(*!
<summary>{attribute 'OPC.UA.DA.Access' := '1'}</summary>
*)

{attribute 'no_explicit_call' := 'do not call this function block directly'}
FUNCTION_BLOCK ABSTRACT ProgramTransition EXTENDS ToolkitObject IMPLEMENTS IAction
VAR_OUTPUT
	
	//Timeout : TIME := T#3S;
END_VAR
VAR
	{attribute 'OPC.UA.DA' := '0'}
	_Busy : BOOL;
	{attribute 'OPC.UA.DA' := '0'}
	_Done : BOOL;
	{attribute 'OPC.UA.DA' := '0'}
	_Error : BOOL;
	{attribute 'OPC.UA.DA' := '0'}
	_StateMachine : REFERENCE TO FiniteStateMachine;
END_VAR

{attribute 'monitoring' := 'call'}
{attribute 'OPC.UA.DA.Property' := '1'}
{attribute 'OPC.UA.DA.Access' := '1'}
PROPERTY Busy : BOOL
GET
Busy := _Busy;
END_GET
END_PROPERTY

METHOD Cancel
IF _Busy THEN
	_Busy := FALSE;	
END_IF
END_METHOD

{attribute 'monitoring' := 'call'}
{attribute 'OPC.UA.DA.Property' := '1'}
{attribute 'OPC.UA.DA.Access' := '1'}
PROPERTY ABSTRACT Cause : STRING
GET
END_GET
END_PROPERTY

{attribute 'monitoring' := 'call'}
{attribute 'OPC.UA.DA.Property' := '1'}
{attribute 'OPC.UA.DA.Access' := '1'}
PROPERTY Done : BOOL
GET
Done := _Done;
END_GET
END_PROPERTY

{attribute 'monitoring' := 'call'}
{attribute 'OPC.UA.DA.Property' := '1'}
{attribute 'OPC.UA.DA.Access' := '1'}
PROPERTY Error : BOOL
GET
Error := _Error;
END_GET
END_PROPERTY

METHOD Execute
_Busy := FALSE;
_Done := TRUE;
_Error := FALSE;
END_METHOD

{attribute 'monitoring' := 'call'}
{attribute 'OPC.UA.DA.Property' := '1'}
{attribute 'OPC.UA.DA.Access' := '1'}
PROPERTY ABSTRACT FromState : STRING
GET
END_GET
END_PROPERTY

METHOD Initialize
VAR_INPUT
	stateMachine : REFERENCE TO FiniteStateMachine;
END_VAR
IF NOT __ISVALIDREF(_StateMachine) THEN
	//exceptionFactory.ThrowException(__POSITION(), "programStateMachine is NULL");
END_IF

_StateMachine REF= stateMachine;
END_METHOD

{attribute 'monitoring' := 'call'}
{attribute 'OPC.UA.DA.Property' := '1'}
{attribute 'OPC.UA.DA.Access' := '1'}
PROPERTY Initialized : BOOL
GET
Initialized := __ISVALIDREF(_StateMachine);
END_GET
END_PROPERTY

{attribute 'monitoring' := 'call'}
PROPERTY LastException : REFERENCE TO Exception
GET
LastException REF= _LastException;
END_GET
END_PROPERTY

{attribute 'monitoring' := 'call'}
{attribute 'OPC.UA.DA.Property' := '1'}
{attribute 'OPC.UA.DA.Access' := '1'}
PROPERTY ABSTRACT Name : STRING
GET
END_GET
END_PROPERTY

METHOD Start
_Busy := FALSE;
_Done := TRUE;
_Error := FALSE;
END_METHOD

{attribute 'monitoring' := 'call'}
{attribute 'OPC.UA.DA.Property' := '1'}
{attribute 'OPC.UA.DA.Access' := '1'}
PROPERTY ABSTRACT ToState : STRING
GET
END_GET
END_PROPERTY

END_FUNCTION_BLOCK

(* stored: Version 1.1.0.1
   POU ProgramTransition: Id {6b59fb44-7d1e-410e-98ab-ba5c7025a4ba}, SpecialFunc None
   Property Busy: Id {b83feb43-f5ff-4bb3-87f5-84ead7a6b586}
   Get Get: Id {ea3ffc98-f880-4a1b-896f-a5358b6fb59b}
   Method Cancel: Id {f4d9f4ec-d47f-4802-b147-e47fb819abd8}
   Property Cause: Id {c9f3fd3d-674d-4611-85bc-8ec662b2c076}
   Get Get: Id {d1aac4fd-1f0a-4a8b-b9e2-9063ada794c0}
   Property Done: Id {c524e9f7-2d5a-4c7e-adac-dc51846488f5}
   Get Get: Id {be929d92-172b-4242-b667-f55e8250fbc4}
   Property Error: Id {fe37c4cb-37ea-43e6-a810-94afe137c611}
   Get Get: Id {4651eb3c-608a-4238-8ae6-8da6f587b31e}
   Method Execute: Id {1585fa56-5dfa-4194-aa2d-51a9ac8d90c2}
   Property FromState: Id {140a3845-da88-47be-b906-08a2791f1ee0}
   Get Get: Id {28420d79-259f-472e-a390-fe4adef5a6f9}
   Method Initialize: Id {5ad33b8d-32bb-4806-b9a7-b1bcb3b6ed0b}
   Property Initialized: Id {806c4f1f-7d5b-45d6-bc3b-59a7e1a8d523}
   Get Get: Id {42fc99a2-a9ac-4723-8140-3ba2ed9bdd1f}
   Property LastException: Id {871d3221-7a43-4236-a533-59853e3634df}
   Get Get: Id {f9397898-9bd2-4c32-90dc-7fd70c10a9d8}
   Property Name: Id {10746e11-2cc2-4dde-b5a1-2e62f40eb852}
   Get Get: Id {802f15a4-5ec9-4633-83ec-1c76cc90efa3}
   Method Start: Id {0f15d627-a5a2-4156-8091-47bce9b97765}
   Property ToState: Id {85b46d87-1f84-4858-9da6-4945abcbfef6}
   Get Get: Id {cd4bad5b-aefa-4f08-8734-511668d57c94} *)
